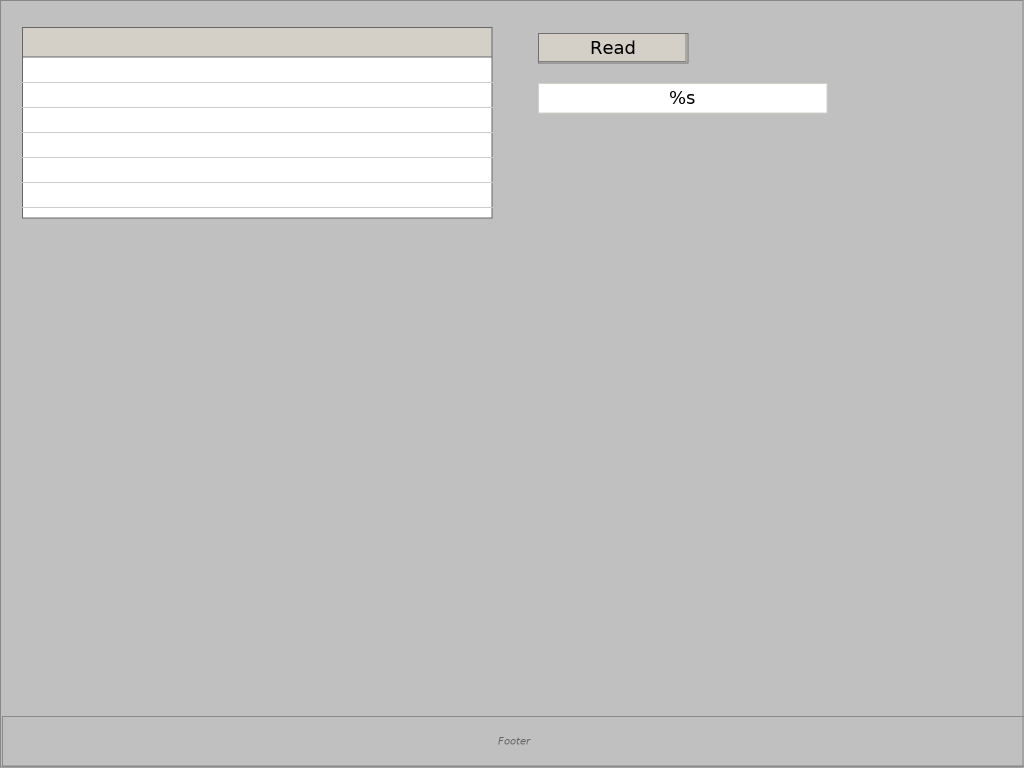
VISUALIZATION Reading  // 1024x768
    Table (22,27 470x191), data array: GVL.readData
        p3854506369: GVL.readData[INDEX].field01
        p1892666644: GVL.readData[INDEX].field02
        p338671338: GVL.readData[INDEX].field03
        p2170511999: GVL.readData[INDEX].field04
        p3723444502: GVL.readData[INDEX].field05
        p2232123230: Field 01
        p511219082: Field 02
        p1755163831: Field 03
        p4092479075: Field 04
        p2237128397: Field 05
    Button (538,33 150x30), "Read"
        tap GVL.readFileNow
    Textfield (538,83 289x30), "%s", text variable: GVL.sFileName
        OnMouseClick: write the text variable via Default
    Frame (2,716 1024x50)
        shows Footer()
END_VISUALIZATION

(* stored: Version 1.1.0.1, ProductVersion 3.1.4024.13
   Visu Reading: Id {9ff5a430-f1a3-4833-bc0c-0721116b3d02} *)
